FUNCTION_BLOCK PWM
VAR_INPUT
END_VAR
VAR_OUTPUT
END_VAR
VAR
	Timer: Timer;
	CurrentDutyCycle: LREAL;
	FPeriod: LREAL;
	FDutyCycle: LREAL;
	FMinValue: LREAL := 0.05; // 5% / 95% min/max value	
END_VAR

PROPERTY DutyCycle : LREAL
GET
DutyCycle := CurrentDutyCycle;
END_GET
SET
VAR
	TimeValue: lreal;	
END_VAR
TimeValue := DutyCycle * Period;
IF (TimeValue < MinValue) THEN
	FDutyCycle := 0;
ELSIF (TimeValue > (Period - MinValue)) THEN
	FDutyCycle := 1;
else
	FDutyCycle := DutyCycle;
END_IF
END_SET
END_PROPERTY

PROPERTY MinValue : LREAL
GET
MinValue := FMinValue;
END_GET
SET
FMinValue := MinValue;
END_SET
END_PROPERTY

PROPERTY Period : LREAL
GET
Period := FPeriod;
END_GET
SET
IF FPeriod <> Period THEN
	FPeriod := Period;
	CurrentDutyCycle := DutyCycle;
	Timer.Restart();
END_IF;
END_SET
END_PROPERTY

METHOD State : BOOL
VAR_INPUT
END_VAR
VAR
	ElapsedTime: LINT;
	Res: BOOL;
END_VAR
ElapsedTime := Timer.ElapsedTime();
IF (ElapsedTime > LREAL_TO_LINT(Period * 1000)) THEN
	ElapsedTime := TRUNC(Period * 1000);
END_IF
Res := ElapsedTime <= LREAL_TO_LINT(CurrentDutyCycle * Period * 1000);
IF (ElapsedTime >= LREAL_TO_LINT(Period * 1000)) THEN
	Timer.Restart();
	CurrentDutyCycle := FDutyCycle;
END_IF;
State := Res;
END_METHOD

END_FUNCTION_BLOCK

(* stored: Version 1.1.0.1, ProductVersion 3.1.4024.3
   POU PWM: Id {9244c080-1b8e-4132-9e3b-730219951ee1}, SpecialFunc None
   Property DutyCycle: Id {781a05bc-2d5d-48b9-a536-eb768315fac6}
   Get Get: Id {cdfd39e1-fb65-43ba-acc4-c08e2cfa70be}
   Set Set: Id {757bccbb-4c3e-490c-89d0-167ae356f8b5}
   Property MinValue: Id {205b2f90-1457-402d-bf51-233e5ce5a668}
   Get Get: Id {fdd455e6-74f6-4e0d-9b8e-7e1c5f1267d0}
   Set Set: Id {879f4242-2c1e-45c3-b1ff-ff74f92fa1c2}
   Property Period: Id {59c802b2-6f6c-4360-b527-3160abaa2dc0}
   Get Get: Id {a36dce81-133c-4e9e-b51f-b1ffcae77743}
   Set Set: Id {5a39a657-4cc8-4a5d-84ae-0d4662c64c7a}
   Method State: Id {d3a21502-b353-457a-9d03-cc872ee3d913} *)
